// TIA Portal V19 export
FUNCTION_BLOCK "HU_Pump"   // FB39, LAD
TITLE = Hydraulic Pump Machine / HYDRAULIC UNIT (MONO-PUMP)
// stored: Access Published, MemoryReserve 100, SetENOAutomatically false
   VAR_INPUT
      AreaInterface : "AreaInterface";
      ZSI : "udt_ZoneSafetyInterface";   // Use only if Safety Cut Off Valve not exist
      DSI : "udt_DeviceSafetyInterface";   // Use only if Safety Cut Off Valve not exist
      DataIn : Struct
         PbStop : Bool;
         PbStart : Bool;
         MainPump_MotorThermalProtection : Bool;
         MainPump_FdbkRunning : Bool;
         SensorPumpFilterClogged : Bool;
      END_STRUCT;
      CIn : Struct
         EnableStopInPhase : Bool;
         EnableStopProgrammed : Bool;
         PumpRunPermitted : Bool;   // From HU_Tank
         EnableCheckFilter : Bool;   // From HU_Tank
         PressureReq : Bool;
      END_STRUCT;
      Config : "HU_Pump_Config";
      Simulation : Bool;
   END_VAR
   VAR_OUTPUT
      MachineInterface : "MachineInterface";
      DataOut : Struct
         KmOilPump : Bool;
         EvAccumulator : Bool;
         EvStandby : Bool;
      END_STRUCT;
      COut : Struct
         CheckNext_Run : Bool;
         CtrlSafe : Bool;
         Standstill : Bool;
         PumpRunning : Bool;
         PressureRunning : Bool;
      END_STRUCT;
   END_VAR
   VAR_IN_OUT
      Par : "HU_Pump_Par";
   END_VAR
   VAR
      M_MainPump : "Motor";
      Ctrl : Struct
         RstAlarms : Bool;
         StopDueDoorOpeningRequest : Bool;
         StopInPhase : Bool;
         StopProgrammed : Bool;
         MainPump_AutStart : Bool;
         MainPump_ManStart : Bool;
      END_STRUCT;
      Sts : Struct
         AlarmsPresence : Bool;
         WarningsPresence : Bool;
         IsStandstill : Bool;
         CndMainPump { ExternalAccessible := 'False'; ExternalVisible := 'False'; ExternalWritable := 'False'} : Bool;
      END_STRUCT;
      HMI : "HU_Pump_HMI";
      Alarm : Struct
         PumpFilterClogged : Bool;
         MainPump : "MotorAlr";
      END_STRUCT;
      Warning : Struct
         NoAutReady : Bool;
      END_STRUCT;
      tonNoPressureReq : IEC_TIMER;
      tonMainPumpInactivity : IEC_TIMER;
      tonDelayPressureStart : IEC_TIMER;
      tonDelayPressureStop : IEC_TIMER;
      tonDelayPressureRunning : IEC_TIMER;
      tonAlrPumpFilterClogged : IEC_TIMER;
      tonNoPendingCmd { S7_SetPoint := 'True'} : IEC_TIMER;
      AckRstAlarms : Bool;
      Pb_Start_PEAux : Bool;
   END_VAR
   VAR_TEMP   // added for the SCL form of the ladder/FBD networks
      _w1 : Bool;
   END_VAR
BEGIN

REGION Network 1 (SCL): Info
   //=============================================================================
   //PM FORMING
   //-----------------------------------------------------------------------------
   // Library: StandardBlocks
   // Tested with: S7-1518TF
   // Engineering: TIA Portal V18
   // Restrictions: -
   // Requirements: S7-1500
   // Functionality: Hydraulic Pump Machine
   //
   // v1.0.0  28/12/2022 
   // v1.1.0  14/02/2023 Simulation added
   // v1.1.1  21/02/2023 DSI Added, for Pump without Safety Cutoff Valve
   // v1.1.2  14/06/2023 Set sensor pump filter clogged NO
   // v1.1.5  29/04/2024 Add reset filter clogged
   //=============================================================================
END_REGION

REGION Network 2 (SCL): Reset alarms command
   #Ctrl.RstAlarms := #AreaInterface.RstAlarms AND NOT #AckRstAlarms; 
   #AckRstAlarms := #AreaInterface.RstAlarms;

   IF #Ctrl.RstAlarms THEN
       #Warning.NoAutReady := FALSE;
       #Alarm.PumpFilterClogged := FALSE;
   END_IF;
END_REGION

REGION Network 3: Alarm pump filter is clogged
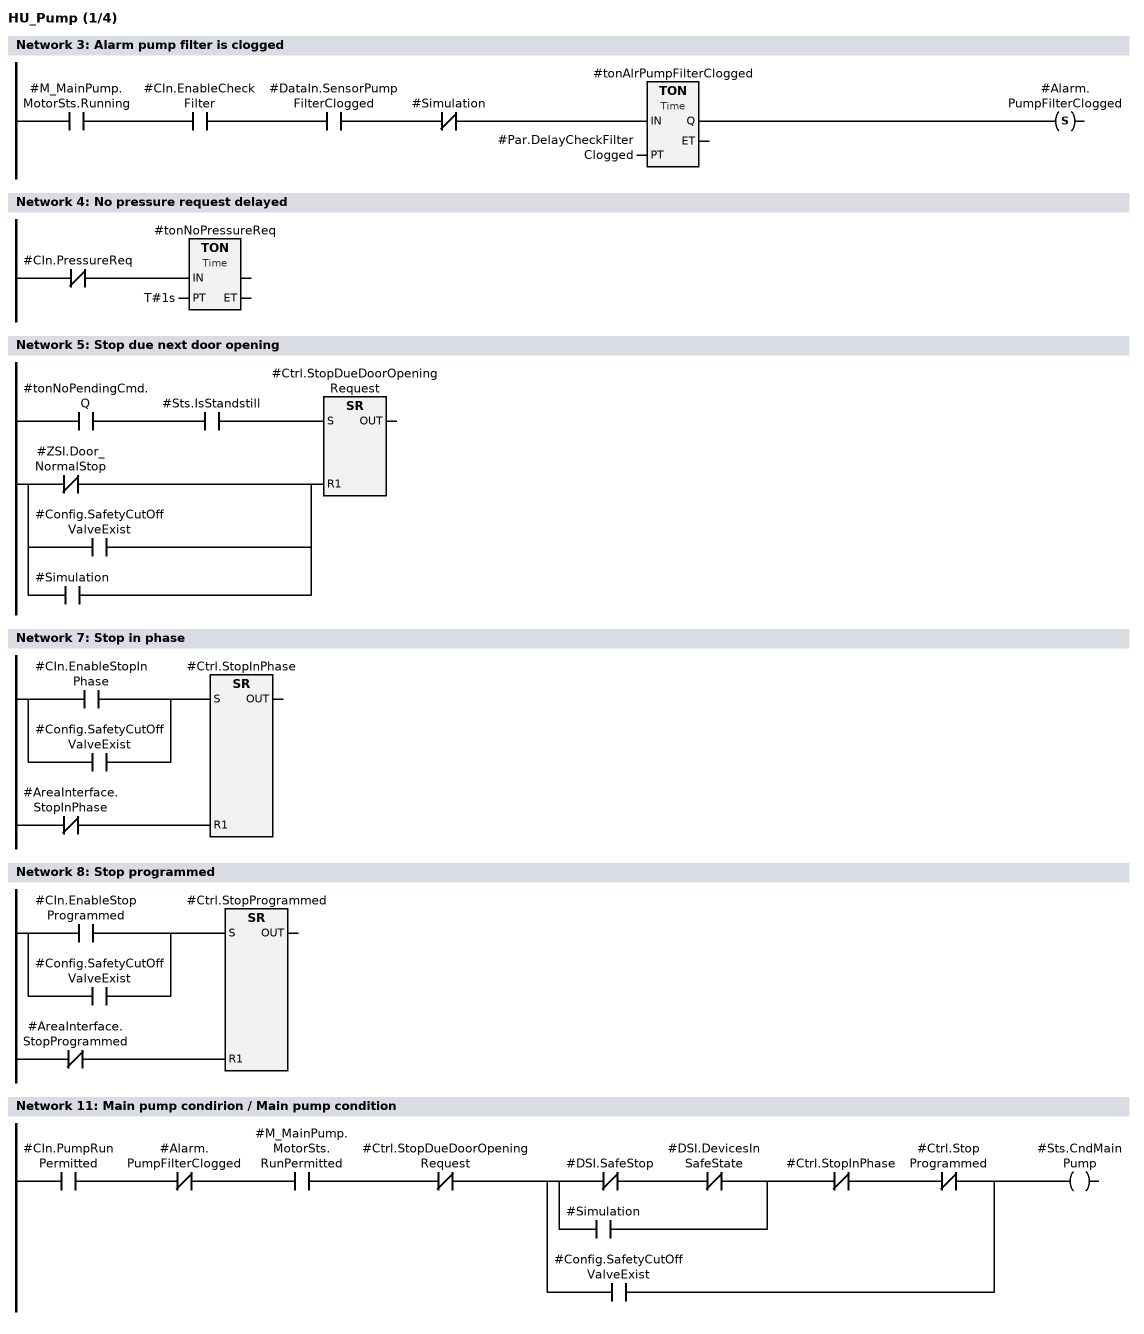
   RUNG wire#powerrail
      Contact( #M_MainPump.MotorSts.Running )
      Contact( #CIn.EnableCheckFilter )
      Contact( #DataIn.SensorPumpFilterClogged )
      I_Contact( #Simulation )
      { S7_Templates := "time_type := Time" } #tonAlrPumpFilterClogged.TON(pt := #Par.DelayCheckFilterClogged, et =>)
      S_Coil( #Alarm.PumpFilterClogged )
   END_RUNG
   // the same network as SCL:
   #tonAlrPumpFilterClogged.TON(IN := #M_MainPump.MotorSts.Running AND #CIn.EnableCheckFilter AND #DataIn.SensorPumpFilterClogged AND NOT #Simulation,
                           PT := #Par.DelayCheckFilterClogged);
   IF #tonAlrPumpFilterClogged.Q THEN #Alarm.PumpFilterClogged := TRUE; END_IF;
END_REGION

REGION Network 4: No pressure request delayed
   RUNG wire#powerrail
      I_Contact( #CIn.PressureReq )
      { S7_Templates := "time_type := Time" } #tonNoPressureReq.TON(pt := T#1s, et =>)
   END_RUNG
   // the same network as SCL:
   #tonNoPressureReq.TON(IN := NOT #CIn.PressureReq, PT := T#1s);
END_REGION

REGION Network 5: Stop due next door opening
   RUNG wire#powerrail
      Contact( #tonNoPendingCmd.Q )
      Contact( #Sts.IsStandstill )
      S_SR(operand := #Ctrl.StopDueDoorOpeningRequest, r1 := wire#w1)
   END_RUNG
   RUNG wire#powerrail
      I_Contact( #ZSI.Door_NormalStop )
   END_RUNG wire#w1
   RUNG wire#powerrail
      Contact( #Config.SafetyCutOffValveExist )
   END_RUNG wire#w1
   RUNG wire#powerrail
      Contact( #Simulation )
   END_RUNG wire#w1
   // the same network as SCL:
   IF #tonNoPendingCmd.Q AND #Sts.IsStandstill THEN
       #Ctrl.StopDueDoorOpeningRequest := TRUE;   // SR flip-flop
   END_IF;
   IF NOT #ZSI.Door_NormalStop OR #Config.SafetyCutOffValveExist OR #Simulation THEN
       #Ctrl.StopDueDoorOpeningRequest := FALSE;
   END_IF;
END_REGION

REGION Network 7: Stop in phase
   RUNG wire#powerrail
      Contact( #CIn.EnableStopInPhase )
      wire#w1
      S_SR(operand := #Ctrl.StopInPhase, r1 := wire#w2)
   END_RUNG
   RUNG wire#powerrail
      Contact( #Config.SafetyCutOffValveExist )
   END_RUNG wire#w1
   RUNG wire#powerrail
      I_Contact( #AreaInterface.StopInPhase )
   END_RUNG wire#w2
   // the same network as SCL:
   IF #CIn.EnableStopInPhase OR #Config.SafetyCutOffValveExist THEN
       #Ctrl.StopInPhase := TRUE;   // SR flip-flop
   END_IF;
   IF NOT #AreaInterface.StopInPhase THEN #Ctrl.StopInPhase := FALSE; END_IF;
END_REGION

REGION Network 8: Stop programmed
   RUNG wire#powerrail
      Contact( #CIn.EnableStopProgrammed )
      wire#w1
      S_SR(operand := #Ctrl.StopProgrammed, r1 := wire#w2)
   END_RUNG
   RUNG wire#powerrail
      Contact( #Config.SafetyCutOffValveExist )
   END_RUNG wire#w1
   RUNG wire#powerrail
      I_Contact( #AreaInterface.StopProgrammed )
   END_RUNG wire#w2
   // the same network as SCL:
   IF #CIn.EnableStopProgrammed OR #Config.SafetyCutOffValveExist THEN
       #Ctrl.StopProgrammed := TRUE;   // SR flip-flop
   END_IF;
   IF NOT #AreaInterface.StopProgrammed THEN #Ctrl.StopProgrammed := FALSE; END_IF;
END_REGION

REGION Network 10: <<< MAIN PUMP >>>
END_REGION

REGION Network 11: Main pump condirion / Main pump condition
   RUNG wire#powerrail
      Contact( #CIn.PumpRunPermitted )
      I_Contact( #Alarm.PumpFilterClogged )
      Contact( #M_MainPump.MotorSts.RunPermitted )
      I_Contact( #Ctrl.StopDueDoorOpeningRequest )
      wire#w1
      I_Contact( #DSI.SafeStop )
      I_Contact( #DSI.DevicesInSafeState )
      wire#w2
      I_Contact( #Ctrl.StopInPhase )
      I_Contact( #Ctrl.StopProgrammed )
      wire#w3
      Coil( #Sts.CndMainPump )
   END_RUNG
   RUNG wire#w1
      Contact( #Simulation )
   END_RUNG wire#w2
   RUNG wire#w1
      Contact( #Config.SafetyCutOffValveExist )
   END_RUNG wire#w3
   // the same network as SCL:
   #Sts.CndMainPump := #CIn.PumpRunPermitted AND NOT #Alarm.PumpFilterClogged AND #M_MainPump.MotorSts.RunPermitted AND NOT #Ctrl.StopDueDoorOpeningRequest AND ((((NOT #DSI.SafeStop AND NOT #DSI.DevicesInSafeState) OR #Simulation) AND NOT #Ctrl.StopInPhase AND NOT #Ctrl.StopProgrammed) OR #Config.SafetyCutOffValveExist);
END_REGION

REGION Network 12: Delay inactivity (no pressure request) / delay inactivity (no pressure request)
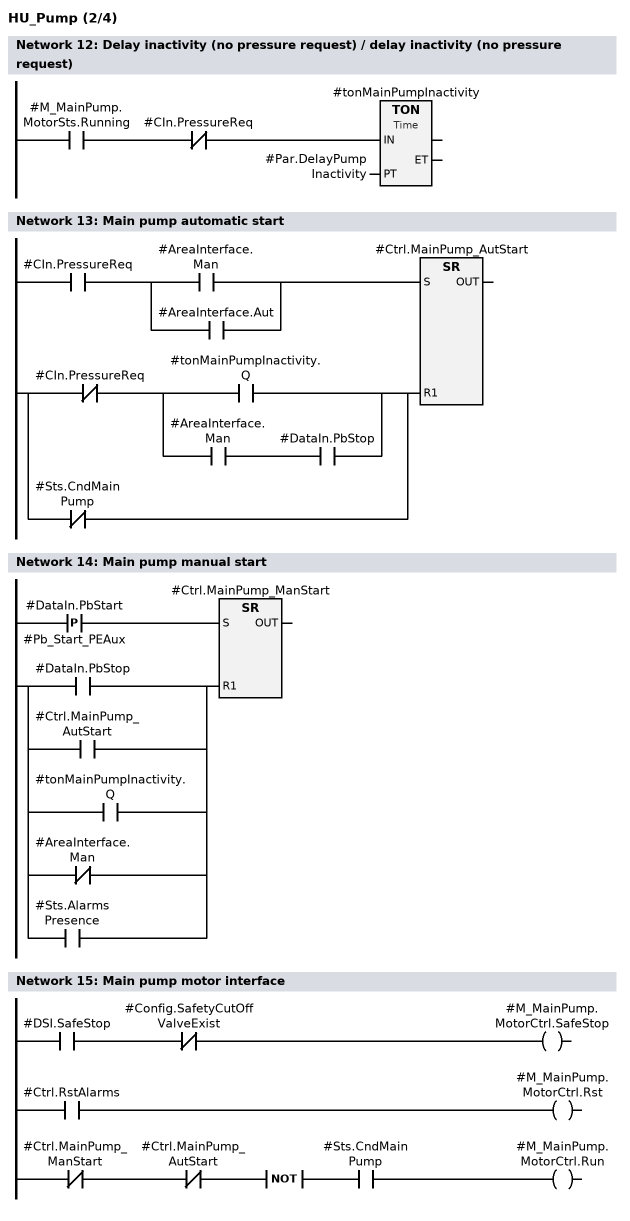
   RUNG wire#powerrail
      Contact( #M_MainPump.MotorSts.Running )
      I_Contact( #CIn.PressureReq )
      { S7_Templates := "time_type := Time" } #tonMainPumpInactivity.TON(pt := #Par.DelayPumpInactivity, et =>)
   END_RUNG
   // the same network as SCL:
   #tonMainPumpInactivity.TON(IN := #M_MainPump.MotorSts.Running AND NOT #CIn.PressureReq,
                           PT := #Par.DelayPumpInactivity);
END_REGION

REGION Network 13: Main pump automatic start
   RUNG wire#powerrail
      Contact( #CIn.PressureReq )
      wire#w1
      Contact( #AreaInterface.Man )
      wire#w2
      S_SR(operand := #Ctrl.MainPump_AutStart, r1 := wire#w4)
   END_RUNG
   RUNG wire#w1
      Contact( #AreaInterface.Aut )
   END_RUNG wire#w2
   RUNG wire#powerrail
      I_Contact( #CIn.PressureReq )
      wire#w3
      Contact( #tonMainPumpInactivity.Q )
   END_RUNG wire#w4
   RUNG wire#w3
      Contact( #AreaInterface.Man )
      Contact( #DataIn.PbStop )
   END_RUNG wire#w4
   RUNG wire#powerrail
      I_Contact( #Sts.CndMainPump )
   END_RUNG wire#w4
   // the same network as SCL:
   IF #CIn.PressureReq AND (#AreaInterface.Man OR #AreaInterface.Aut) THEN
       #Ctrl.MainPump_AutStart := TRUE;   // SR flip-flop
   END_IF;
   IF (NOT #CIn.PressureReq AND (#tonMainPumpInactivity.Q OR (#AreaInterface.Man AND #DataIn.PbStop))) OR NOT #Sts.CndMainPump THEN
       #Ctrl.MainPump_AutStart := FALSE;
   END_IF;
END_REGION

REGION Network 14: Main pump manual start
   RUNG wire#powerrail
      P_Contact(operand := #DataIn.PbStart, bit := #Pb_Start_PEAux)
      S_SR(operand := #Ctrl.MainPump_ManStart, r1 := wire#w1)
   END_RUNG
   RUNG wire#powerrail
      Contact( #DataIn.PbStop )
   END_RUNG wire#w1
   RUNG wire#powerrail
      Contact( #Ctrl.MainPump_AutStart )
   END_RUNG wire#w1
   RUNG wire#powerrail
      Contact( #tonMainPumpInactivity.Q )
   END_RUNG wire#w1
   RUNG wire#powerrail
      I_Contact( #AreaInterface.Man )
   END_RUNG wire#w1
   RUNG wire#powerrail
      Contact( #Sts.AlarmsPresence )
   END_RUNG wire#w1
   // the same network as SCL:
   #_w1 := #DataIn.PbStart AND NOT #Pb_Start_PEAux;   // rising edge of #DataIn.PbStart
   #Pb_Start_PEAux := #DataIn.PbStart;
   IF #_w1 THEN
       #Ctrl.MainPump_ManStart := TRUE;   // SR flip-flop
   END_IF;
   IF #DataIn.PbStop OR #Ctrl.MainPump_AutStart OR #tonMainPumpInactivity.Q OR NOT #AreaInterface.Man OR #Sts.AlarmsPresence THEN
       #Ctrl.MainPump_ManStart := FALSE;
   END_IF;
END_REGION

REGION Network 15: Main pump motor interface
   RUNG wire#powerrail
      Contact( #DSI.SafeStop )
      I_Contact( #Config.SafetyCutOffValveExist )
      Coil( #M_MainPump.MotorCtrl.SafeStop )
   END_RUNG
   RUNG wire#powerrail
      Contact( #Ctrl.RstAlarms )
      Coil( #M_MainPump.MotorCtrl.Rst )
   END_RUNG
   RUNG wire#powerrail
      I_Contact( #Ctrl.MainPump_ManStart )
      I_Contact( #Ctrl.MainPump_AutStart )
      Not()
      Contact( #Sts.CndMainPump )
      Coil( #M_MainPump.MotorCtrl.Run )
   END_RUNG
   // the same network as SCL:
   #M_MainPump.MotorCtrl.SafeStop := #DSI.SafeStop AND NOT #Config.SafetyCutOffValveExist;
   #M_MainPump.MotorCtrl.Rst := #Ctrl.RstAlarms;
   #M_MainPump.MotorCtrl.Run := NOT (NOT #Ctrl.MainPump_ManStart AND NOT #Ctrl.MainPump_AutStart) AND #Sts.CndMainPump;
END_REGION

REGION Network 16: Main pump motor manager
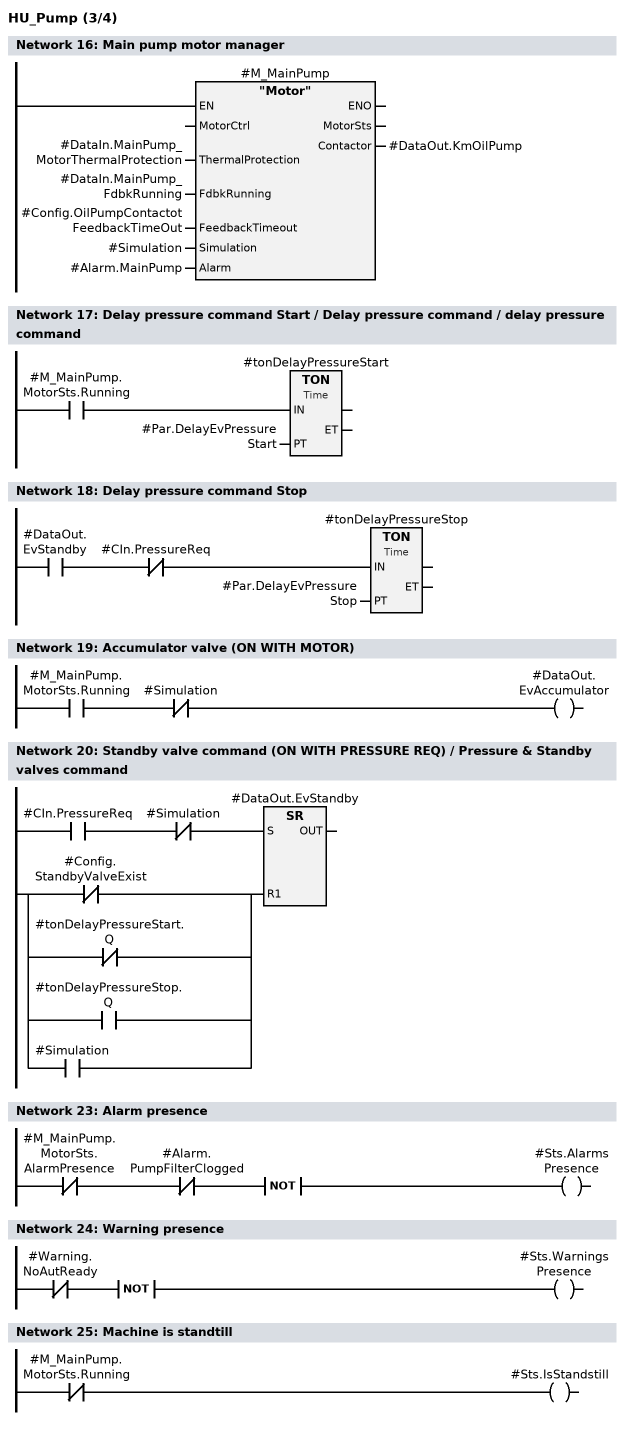
   RUNG wire#powerrail
      #M_MainPump(MotorCtrl :=, ThermalProtection := #DataIn.MainPump_MotorThermalProtection, FdbkRunning := #DataIn.MainPump_FdbkRunning, FeedbackTimeout := #Config.OilPumpContactotFeedbackTimeOut, Simulation := #Simulation, Alarm := #Alarm.MainPump, MotorSts =>, Contactor => #DataOut.KmOilPump)
   END_RUNG
   // the same network as SCL:
   #M_MainPump(ThermalProtection := #DataIn.MainPump_MotorThermalProtection,   // "Motor"
               FdbkRunning := #DataIn.MainPump_FdbkRunning,
               FeedbackTimeout := #Config.OilPumpContactotFeedbackTimeOut,
               Simulation := #Simulation,
               Alarm := #Alarm.MainPump,
               Contactor => #DataOut.KmOilPump);
END_REGION

REGION Network 17: Delay pressure command Start / Delay pressure command / delay pressure command
   RUNG wire#powerrail
      Contact( #M_MainPump.MotorSts.Running )
      { S7_Templates := "time_type := Time" } #tonDelayPressureStart.TON(pt := #Par.DelayEvPressureStart, et =>)
   END_RUNG
   // the same network as SCL:
   #tonDelayPressureStart.TON(IN := #M_MainPump.MotorSts.Running, PT := #Par.DelayEvPressureStart);
END_REGION

REGION Network 18: Delay pressure command Stop
   RUNG wire#powerrail
      Contact( #DataOut.EvStandby )
      I_Contact( #CIn.PressureReq )
      { S7_Templates := "time_type := Time" } #tonDelayPressureStop.TON(pt := #Par.DelayEvPressureStop, et =>)
   END_RUNG
   // the same network as SCL:
   #tonDelayPressureStop.TON(IN := #DataOut.EvStandby AND NOT #CIn.PressureReq, PT := #Par.DelayEvPressureStop);
END_REGION

REGION Network 19: Accumulator valve (ON WITH MOTOR)
   RUNG wire#powerrail
      Contact( #M_MainPump.MotorSts.Running )
      I_Contact( #Simulation )
      Coil( #DataOut.EvAccumulator )
   END_RUNG
   // the same network as SCL:
   #DataOut.EvAccumulator := #M_MainPump.MotorSts.Running AND NOT #Simulation;
END_REGION

REGION Network 20: Standby valve command (ON WITH PRESSURE REQ) / Pressure & Standby valves command
   RUNG wire#powerrail
      Contact( #CIn.PressureReq )
      I_Contact( #Simulation )
      S_SR(operand := #DataOut.EvStandby, r1 := wire#w1)
   END_RUNG
   RUNG wire#powerrail
      I_Contact( #Config.StandbyValveExist )
   END_RUNG wire#w1
   RUNG wire#powerrail
      I_Contact( #tonDelayPressureStart.Q )
   END_RUNG wire#w1
   RUNG wire#powerrail
      Contact( #tonDelayPressureStop.Q )
   END_RUNG wire#w1
   RUNG wire#powerrail
      Contact( #Simulation )
   END_RUNG wire#w1
   // the same network as SCL:
   IF #CIn.PressureReq AND NOT #Simulation THEN
       #DataOut.EvStandby := TRUE;   // SR flip-flop
   END_IF;
   IF NOT #Config.StandbyValveExist OR NOT #tonDelayPressureStart.Q OR #tonDelayPressureStop.Q OR #Simulation THEN
       #DataOut.EvStandby := FALSE;
   END_IF;
END_REGION

REGION Network 22: <<<< + >>>>>>>
END_REGION

REGION Network 23: Alarm presence
   RUNG wire#powerrail
      I_Contact( #M_MainPump.MotorSts.AlarmPresence )
      I_Contact( #Alarm.PumpFilterClogged )
      Not()
      Coil( #Sts.AlarmsPresence )
   END_RUNG
   // the same network as SCL:
   #Sts.AlarmsPresence := NOT (NOT #M_MainPump.MotorSts.AlarmPresence AND NOT #Alarm.PumpFilterClogged);
END_REGION

REGION Network 24: Warning presence
   RUNG wire#powerrail
      I_Contact( #Warning.NoAutReady )
      Not()
      Coil( #Sts.WarningsPresence )
   END_RUNG
   // the same network as SCL:
   #Sts.WarningsPresence := NOT (NOT #Warning.NoAutReady);
END_REGION

REGION Network 25: Machine is standtill
   RUNG wire#powerrail
      I_Contact( #M_MainPump.MotorSts.Running )
      Coil( #Sts.IsStandstill )
   END_RUNG
   // the same network as SCL:
   #Sts.IsStandstill := NOT #M_MainPump.MotorSts.Running;
END_REGION

REGION Network 26: No Pending command
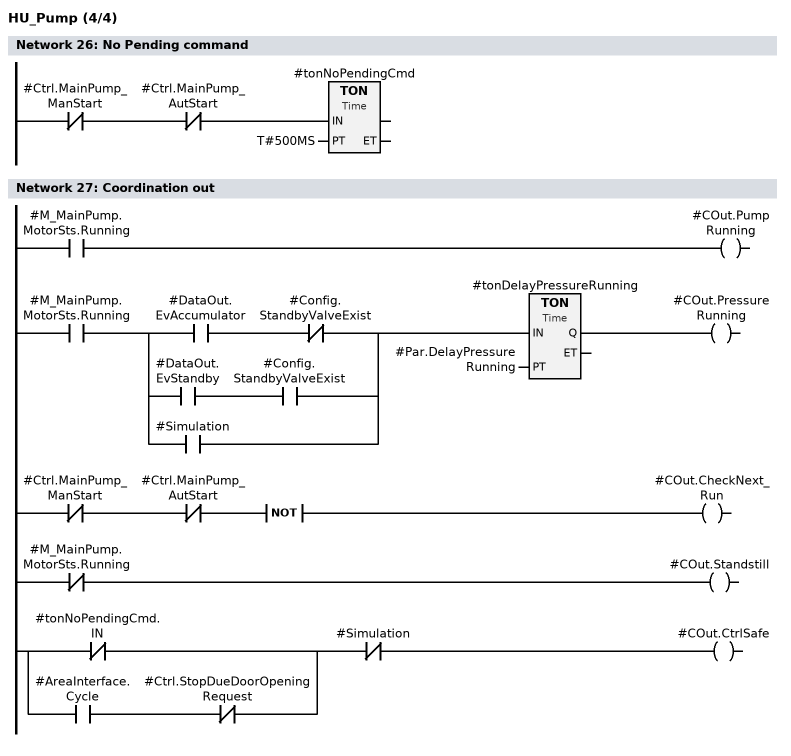
   RUNG wire#powerrail
      I_Contact( #Ctrl.MainPump_ManStart )
      I_Contact( #Ctrl.MainPump_AutStart )
      { S7_Templates := "time_type := Time" } #tonNoPendingCmd.TON(pt := T#500MS, et =>)
   END_RUNG
   // the same network as SCL:
   #tonNoPendingCmd.TON(IN := NOT #Ctrl.MainPump_ManStart AND NOT #Ctrl.MainPump_AutStart, PT := T#500MS);
END_REGION

REGION Network 27: Coordination out
   RUNG wire#powerrail
      Contact( #M_MainPump.MotorSts.Running )
      Coil( #COut.PumpRunning )
   END_RUNG
   RUNG wire#powerrail
      Contact( #M_MainPump.MotorSts.Running )
      wire#w1
      Contact( #DataOut.EvAccumulator )
      I_Contact( #Config.StandbyValveExist )
      wire#w2
      { S7_Templates := "time_type := Time" } #tonDelayPressureRunning.TON(pt := #Par.DelayPressureRunning, et =>)
      Coil( #COut.PressureRunning )
   END_RUNG
   RUNG wire#w1
      Contact( #DataOut.EvStandby )
      Contact( #Config.StandbyValveExist )
   END_RUNG wire#w2
   RUNG wire#w1
      Contact( #Simulation )
   END_RUNG wire#w2
   RUNG wire#powerrail
      I_Contact( #Ctrl.MainPump_ManStart )
      I_Contact( #Ctrl.MainPump_AutStart )
      Not()
      Coil( #COut.CheckNext_Run )
   END_RUNG
   RUNG wire#powerrail
      I_Contact( #M_MainPump.MotorSts.Running )
      Coil( #COut.Standstill )
   END_RUNG
   RUNG wire#powerrail
      I_Contact( #tonNoPendingCmd.IN )
      wire#w3
      I_Contact( #Simulation )
      Coil( #COut.CtrlSafe )
   END_RUNG
   RUNG wire#powerrail
      Contact( #AreaInterface.Cycle )
      I_Contact( #Ctrl.StopDueDoorOpeningRequest )
   END_RUNG wire#w3
   // the same network as SCL:
   #COut.PumpRunning := #M_MainPump.MotorSts.Running;
   #tonDelayPressureRunning.TON(IN := #M_MainPump.MotorSts.Running AND ((#DataOut.EvAccumulator AND NOT #Config.StandbyValveExist) OR (#DataOut.EvStandby AND #Config.StandbyValveExist) OR #Simulation),
                           PT := #Par.DelayPressureRunning);
   #COut.PressureRunning := #tonDelayPressureRunning.Q;
   #COut.CheckNext_Run := NOT (NOT #Ctrl.MainPump_ManStart AND NOT #Ctrl.MainPump_AutStart);
   #COut.Standstill := NOT #M_MainPump.MotorSts.Running;
   #COut.CtrlSafe := (NOT #tonNoPendingCmd.IN OR (#AreaInterface.Cycle AND NOT #Ctrl.StopDueDoorOpeningRequest)) AND NOT #Simulation;
END_REGION

REGION Network 28 (SCL): HMI
   #HMI.Alarm := #Sts.AlarmsPresence;
   #HMI.ManStart := #Ctrl.MainPump_ManStart;
   #HMI.PumpRunning := #COut.PumpRunning;
   #HMI.PressureRunning := #COut.PressureRunning;
END_REGION

REGION Network 29 (SCL): Collect machine to area interface
   // Status machine ready
   #MachineInterface.AutReady := #AreaInterface.Aut AND NOT #Sts.AlarmsPresence;
   // Status machine aborting
   #MachineInterface.Aborting := #Sts.AlarmsPresence;
   // Status Ack Stop in phase
   #MachineInterface.AckStopInPhase := #Ctrl.StopInPhase AND (#Sts.IsStandstill OR #Config.SafetyCutOffValveExist);
   // Status Ack Stop programmed
   #MachineInterface.AckStopProgrammed := #Ctrl.StopProgrammed AND (#Sts.IsStandstill OR #Config.SafetyCutOffValveExist);
   // Status Motion standtill
   #MachineInterface.MotionsStandStill := #Sts.IsStandstill;
   // Status Alarm presence
   #MachineInterface.AlarmsPresence := #Sts.AlarmsPresence;
   // Status Warning presence
   #MachineInterface.WarningPresence := #Sts.WarningsPresence;

   // Warning machine not automatic ready
   IF #AreaInterface.CheckAutReady AND NOT #MachineInterface.AutReady THEN
     #Warning.NoAutReady := false;
   END_IF;
END_REGION
END_FUNCTION_BLOCK
